// TIA Portal V20 export
FUNCTION "CallEnergyMeter" : Void   // FC9, LAD
TITLE = CALL_AIEnergyMeter_FC
AUTHOR : SICAR
FAMILY : Energy
VERSION : 1.0
// This block calls the blocks for the AI-Energy-management.
// For more informations see SICAR userdefined documentation / SICAR online-help.
// stored: IsIECCheckEnabled true, SetENOAutomatically true
   VAR_TEMP
      tempCommResourceCounter : Int;   // für FB-Aufruf: E2M_1500_AIEnergyMeter_DRV
      tempBitsHmi : "typeEnMeterBits";   // für FB-Aufruf: E2M_1500_AIEnergyMeter_DRV
   END_VAR
   // Ret_Val : Ret_Val
BEGIN

REGION Network 1: ChangeLog
   // SIEMENS AG / (c)Copyright 2023
   // ------------------------------------------------------------------------------
   // Title:            CallEnergyMeter (FC9)
   // Comment/Function: This block calls the blocks for the AI-Energy-management.
   // Library/Family:   Automation Framework
   // Author:           Siemens Digital Industry
   // Tested with:      ---
   // Engineering:      TIA Portal V19
   // Restrictions:     -
   // Requirements:     ---
   // ------------------------------------------------------------------------------
   // Change log table:
   // Version  | Date       | Expert in charge       | Changes applied
   // ---------|------------|------------------------|------------------------------
   // 05.00.00 | 01.09.2023 | SICAR
   //                         First released version
END_REGION

REGION Network 2: AI_EnergyMeter 1
   // Call of E2MenergyMeterDrv FB
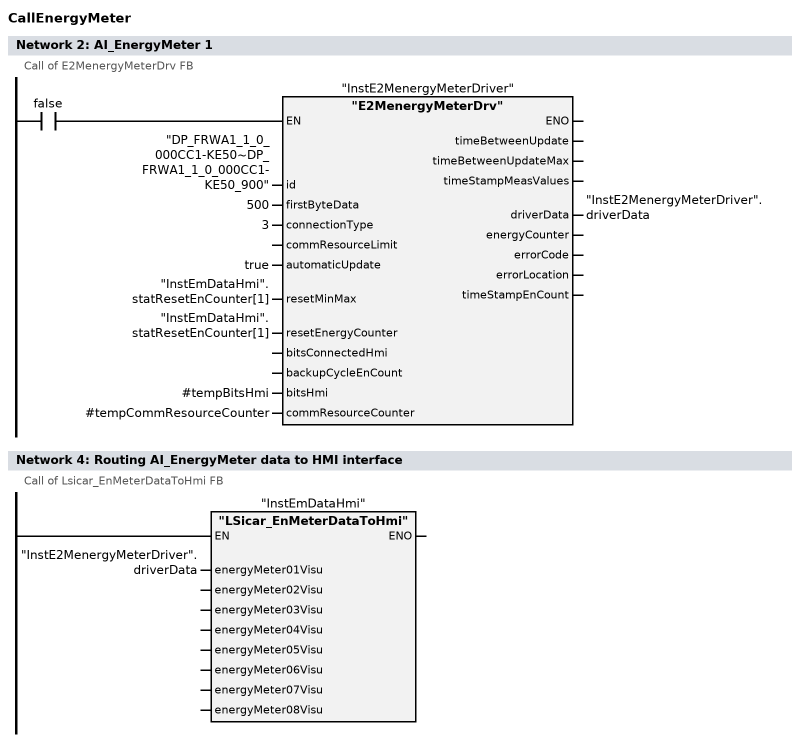
   RUNG wire#powerrail
      Contact( false )
      "InstE2MenergyMeterDriver"(id := "DP_FRWA1_1_0_000CC1-KE50~DP_FRWA1_1_0_000CC1-KE50_900", firstByteData := 500, connectionType := 3, commResourceLimit :=, automaticUpdate := true, resetMinMax := "InstEmDataHmi".statResetEnCounter[1], resetEnergyCounter := "InstEmDataHmi".statResetEnCounter[1], bitsConnectedHmi :=, backupCycleEnCount :=, bitsHmi := #tempBitsHmi, commResourceCounter := #tempCommResourceCounter, timeBetweenUpdate =>, timeBetweenUpdateMax =>, timeStampMeasValues =>, driverData => "InstE2MenergyMeterDriver".driverData, energyCounter =>, errorCode =>, errorLocation =>, timeStampEnCount =>)
   END_RUNG
   // the same network as SCL:
   IF false THEN
       "InstE2MenergyMeterDriver"(id := "DP_FRWA1_1_0_000CC1-KE50~DP_FRWA1_1_0_000CC1-KE50_900",   // "E2MenergyMeterDrv"
                               firstByteData := 500,
                               connectionType := 3,
                               automaticUpdate := true,
                               resetMinMax := "InstEmDataHmi".statResetEnCounter[1],
                               resetEnergyCounter := "InstEmDataHmi".statResetEnCounter[1],
                               bitsHmi := #tempBitsHmi,
                               commResourceCounter := #tempCommResourceCounter,
                               driverData => "InstE2MenergyMeterDriver".driverData);
   END_IF;
END_REGION

REGION Network 3 (SCL): Power meter

   // Voltage L-N
   "InstE2MenergyMeterDriver".driverData.uL1 := "PAC3220InPut"."Voltage_L1-N";
   "InstE2MenergyMeterDriver".driverData.uL2 := "PAC3220InPut"."Voltage_L2-N";
   "InstE2MenergyMeterDriver".driverData.uL3 := "PAC3220InPut"."Voltage_L3-N";
   "InstE2MenergyMeterDriver".driverData.uPhNaverage :=
   ("InstE2MenergyMeterDriver".driverData.uL1 + "InstE2MenergyMeterDriver".driverData.uL2 + "InstE2MenergyMeterDriver".driverData.uL3) / 3.0;

   IF "InstE2MenergyMeterDriver".driverData.uL1 < "InstE2MenergyMeterDriver".driverData.uL1Min OR "InstE2MenergyMeterDriver".driverData.uL1Min = 0.0 THEN
       "InstE2MenergyMeterDriver".driverData.uL1Min := "InstE2MenergyMeterDriver".driverData.uL1;
   END_IF;
   IF "InstE2MenergyMeterDriver".driverData.uL1 > "InstE2MenergyMeterDriver".driverData.uL1Max OR "InstE2MenergyMeterDriver".driverData.uL1Max = 0.0 THEN
       "InstE2MenergyMeterDriver".driverData.uL1Max := "InstE2MenergyMeterDriver".driverData.uL1;
   END_IF;

   IF "InstE2MenergyMeterDriver".driverData.uL2 < "InstE2MenergyMeterDriver".driverData.uL2Min OR "InstE2MenergyMeterDriver".driverData.uL2Min = 0.0 THEN
       "InstE2MenergyMeterDriver".driverData.uL2Min := "InstE2MenergyMeterDriver".driverData.uL2;
   END_IF;
   IF "InstE2MenergyMeterDriver".driverData.uL2 > "InstE2MenergyMeterDriver".driverData.uL2Max OR "InstE2MenergyMeterDriver".driverData.uL2Max = 0.0 THEN
       "InstE2MenergyMeterDriver".driverData.uL2Max := "InstE2MenergyMeterDriver".driverData.uL2;
   END_IF;

   IF "InstE2MenergyMeterDriver".driverData.uL3 < "InstE2MenergyMeterDriver".driverData.uL3Min OR "InstE2MenergyMeterDriver".driverData.uL3Min = 0.0 THEN
       "InstE2MenergyMeterDriver".driverData.uL3Min := "InstE2MenergyMeterDriver".driverData.uL3;
   END_IF;
   IF "InstE2MenergyMeterDriver".driverData.uL3 > "InstE2MenergyMeterDriver".driverData.uL3Max OR "InstE2MenergyMeterDriver".driverData.uL3Max = 0.0 THEN
       "InstE2MenergyMeterDriver".driverData.uL3Max := "InstE2MenergyMeterDriver".driverData.uL3;
   END_IF;

   IF "InstE2MenergyMeterDriver".driverData.uPhNaverage < "InstE2MenergyMeterDriver".driverData.uPhNaverageMin OR "InstE2MenergyMeterDriver".driverData.uPhNaverageMin = 0.0 THEN
       "InstE2MenergyMeterDriver".driverData.uPhNaverageMin := "InstE2MenergyMeterDriver".driverData.uPhNaverage;
   END_IF;
   IF "InstE2MenergyMeterDriver".driverData.uPhNaverage > "InstE2MenergyMeterDriver".driverData.uPhNaverageMax OR "InstE2MenergyMeterDriver".driverData.uPhNaverageMax = 0.0 THEN
       "InstE2MenergyMeterDriver".driverData.uPhNaverageMax := "InstE2MenergyMeterDriver".driverData.uPhNaverage;
   END_IF;

   // Voltage L-L
   "InstE2MenergyMeterDriver".driverData.uL1L2 := "PAC3220InPut"."Voltage_L1-L2";
   "InstE2MenergyMeterDriver".driverData.uL2L3 := "PAC3220InPut"."Voltage_L2-L3";
   "InstE2MenergyMeterDriver".driverData.uL3L1 := "PAC3220InPut"."Voltage_L3-L1";
   "InstE2MenergyMeterDriver".driverData.uPhPhAverage :=
   ("InstE2MenergyMeterDriver".driverData.uL1L2 + "InstE2MenergyMeterDriver".driverData.uL2L3 + "InstE2MenergyMeterDriver".driverData.uL3L1) / 3.0;

   IF "InstE2MenergyMeterDriver".driverData.uL1L2 < "InstE2MenergyMeterDriver".driverData.uL1L2Min OR "InstE2MenergyMeterDriver".driverData.uL1L2Min = 0.0 THEN
       "InstE2MenergyMeterDriver".driverData.uL1L2Min := "InstE2MenergyMeterDriver".driverData.uL1L2;
   END_IF;
   IF "InstE2MenergyMeterDriver".driverData.uL1L2 > "InstE2MenergyMeterDriver".driverData.uL1L2Max OR "InstE2MenergyMeterDriver".driverData.uL1L2Max = 0.0 THEN
       "InstE2MenergyMeterDriver".driverData.uL1L2Max := "InstE2MenergyMeterDriver".driverData.uL1L2;
   END_IF;

   IF "InstE2MenergyMeterDriver".driverData.uL2L3 < "InstE2MenergyMeterDriver".driverData.uL2L3Min OR "InstE2MenergyMeterDriver".driverData.uL2L3Min = 0.0 THEN
       "InstE2MenergyMeterDriver".driverData.uL2L3Min := "InstE2MenergyMeterDriver".driverData.uL2L3;
   END_IF;
   IF "InstE2MenergyMeterDriver".driverData.uL2L3 > "InstE2MenergyMeterDriver".driverData.uL2L3Max OR "InstE2MenergyMeterDriver".driverData.uL2L3Max = 0.0 THEN
       "InstE2MenergyMeterDriver".driverData.uL2L3Max := "InstE2MenergyMeterDriver".driverData.uL2L3;
   END_IF;

   IF "InstE2MenergyMeterDriver".driverData.uL3L1 < "InstE2MenergyMeterDriver".driverData.uL3L1Min OR "InstE2MenergyMeterDriver".driverData.uL3L1Min = 0.0 THEN
       "InstE2MenergyMeterDriver".driverData.uL3L1Min := "InstE2MenergyMeterDriver".driverData.uL3L1;
   END_IF;
   IF "InstE2MenergyMeterDriver".driverData.uL3L1 > "InstE2MenergyMeterDriver".driverData.uL3L1Max OR "InstE2MenergyMeterDriver".driverData.uL3L1Max = 0.0 THEN
       "InstE2MenergyMeterDriver".driverData.uL3L1Max := "InstE2MenergyMeterDriver".driverData.uL3L1;
   END_IF;

   IF "InstE2MenergyMeterDriver".driverData.uPhPhAverage < "InstE2MenergyMeterDriver".driverData.uPhPhAverageMin OR "InstE2MenergyMeterDriver".driverData.uPhPhAverageMin = 0.0 THEN
       "InstE2MenergyMeterDriver".driverData.uPhPhAverageMin := "InstE2MenergyMeterDriver".driverData.uPhPhAverage;
   END_IF;
   IF "InstE2MenergyMeterDriver".driverData.uPhPhAverage > "InstE2MenergyMeterDriver".driverData.uPhPhAverageMax OR "InstE2MenergyMeterDriver".driverData.uPhPhAverageMax = 0.0THEN
       "InstE2MenergyMeterDriver".driverData.uPhPhAverageMax := "InstE2MenergyMeterDriver".driverData.uPhPhAverage;
   END_IF;

   // Current
   "InstE2MenergyMeterDriver".driverData.iL1 := "PAC3220InPut".Current_L1;
   "InstE2MenergyMeterDriver".driverData.iL2 := "PAC3220InPut".Current_L2;
   "InstE2MenergyMeterDriver".driverData.iL3 := "PAC3220InPut".Current_L3;
   "InstE2MenergyMeterDriver".driverData.iAverage := "PAC3220InPut"."3-phase_average_current";

   IF "InstE2MenergyMeterDriver".driverData.iL1 < "InstE2MenergyMeterDriver".driverData.iL1Min OR "InstE2MenergyMeterDriver".driverData.iL1Min = 0.0 THEN
       "InstE2MenergyMeterDriver".driverData.iL1Min := "InstE2MenergyMeterDriver".driverData.iL1;
   END_IF;
   IF "InstE2MenergyMeterDriver".driverData.iL1 > "InstE2MenergyMeterDriver".driverData.iL1Max OR "InstE2MenergyMeterDriver".driverData.iL1Max = 0.0 THEN
       "InstE2MenergyMeterDriver".driverData.iL1Max := "InstE2MenergyMeterDriver".driverData.iL1;
   END_IF;

   IF "InstE2MenergyMeterDriver".driverData.iL2 < "InstE2MenergyMeterDriver".driverData.iL2Min OR "InstE2MenergyMeterDriver".driverData.iL2Min = 0.0 THEN
       "InstE2MenergyMeterDriver".driverData.iL2Min := "InstE2MenergyMeterDriver".driverData.iL2;
   END_IF;
   IF "InstE2MenergyMeterDriver".driverData.iL2 > "InstE2MenergyMeterDriver".driverData.iL2Max OR "InstE2MenergyMeterDriver".driverData.iL2Max = 0.0 THEN
       "InstE2MenergyMeterDriver".driverData.iL2Max := "InstE2MenergyMeterDriver".driverData.iL2;
   END_IF;

   IF "InstE2MenergyMeterDriver".driverData.iL3 < "InstE2MenergyMeterDriver".driverData.iL3Min OR "InstE2MenergyMeterDriver".driverData.iL3Min = 0.0 THEN
       "InstE2MenergyMeterDriver".driverData.iL3Min := "InstE2MenergyMeterDriver".driverData.iL3;
   END_IF;
   IF "InstE2MenergyMeterDriver".driverData.iL3 > "InstE2MenergyMeterDriver".driverData.iL3Max OR "InstE2MenergyMeterDriver".driverData.iL3Max = 0.0 THEN
       "InstE2MenergyMeterDriver".driverData.iL3Max := "InstE2MenergyMeterDriver".driverData.iL3;
   END_IF;

   IF "InstE2MenergyMeterDriver".driverData.iAverage < "InstE2MenergyMeterDriver".driverData.iAverageMin OR "InstE2MenergyMeterDriver".driverData.iAverageMin = 0.0 THEN
       "InstE2MenergyMeterDriver".driverData.iAverageMin := "InstE2MenergyMeterDriver".driverData.iAverage;
   END_IF;
   IF "InstE2MenergyMeterDriver".driverData.iAverage > "InstE2MenergyMeterDriver".driverData.iAverageMax OR "InstE2MenergyMeterDriver".driverData.iAverageMax = 0.0THEN
       "InstE2MenergyMeterDriver".driverData.iAverageMax := "InstE2MenergyMeterDriver".driverData.iAverage;
   END_IF;

   // Power factor
   "InstE2MenergyMeterDriver".driverData.cosL1 := "PAC3220InPut".Power_factor_L1;
   "InstE2MenergyMeterDriver".driverData.cosL2 := "PAC3220InPut".Power_factor_L2;
   "InstE2MenergyMeterDriver".driverData.cosL3 := "PAC3220InPut".Power_factor_L3;
   "InstE2MenergyMeterDriver".driverData.cosAverage := "PAC3220InPut".Total_power_factor;

   IF "InstE2MenergyMeterDriver".driverData.cosL1 < "InstE2MenergyMeterDriver".driverData.cosL1Min OR "InstE2MenergyMeterDriver".driverData.cosL1Min = 0.0 THEN
       "InstE2MenergyMeterDriver".driverData.cosL1Min := "InstE2MenergyMeterDriver".driverData.cosL1;
   END_IF;
   IF "InstE2MenergyMeterDriver".driverData.cosL1 > "InstE2MenergyMeterDriver".driverData.cosL1Max THEN
       "InstE2MenergyMeterDriver".driverData.cosL1Max := "InstE2MenergyMeterDriver".driverData.cosL1;
   END_IF;

   IF "InstE2MenergyMeterDriver".driverData.cosL2 < "InstE2MenergyMeterDriver".driverData.cosL2Min OR "InstE2MenergyMeterDriver".driverData.cosL2Min = 0.0 THEN
       "InstE2MenergyMeterDriver".driverData.cosL2Min := "InstE2MenergyMeterDriver".driverData.cosL2;
   END_IF;
   IF "InstE2MenergyMeterDriver".driverData.cosL2 > "InstE2MenergyMeterDriver".driverData.cosL2Max OR "InstE2MenergyMeterDriver".driverData.cosL2Max = 0.0 THEN
       "InstE2MenergyMeterDriver".driverData.cosL2Max := "InstE2MenergyMeterDriver".driverData.cosL2;
   END_IF;

   IF "InstE2MenergyMeterDriver".driverData.cosL3 < "InstE2MenergyMeterDriver".driverData.cosL3Min OR "InstE2MenergyMeterDriver".driverData.cosL3Min = 0.0 THEN
       "InstE2MenergyMeterDriver".driverData.cosL3Min := "InstE2MenergyMeterDriver".driverData.cosL3;
   END_IF;
   IF "InstE2MenergyMeterDriver".driverData.cosL3 > "InstE2MenergyMeterDriver".driverData.cosL3Max OR "InstE2MenergyMeterDriver".driverData.cosL3Max = 0.0THEN
       "InstE2MenergyMeterDriver".driverData.cosL3Max := "InstE2MenergyMeterDriver".driverData.cosL3;
   END_IF;

   IF "InstE2MenergyMeterDriver".driverData.cosAverage < "InstE2MenergyMeterDriver".driverData.cosAverageMin OR "InstE2MenergyMeterDriver".driverData.cosAverageMin = 0.0 THEN
       "InstE2MenergyMeterDriver".driverData.cosAverageMin := "InstE2MenergyMeterDriver".driverData.cosAverage;
   END_IF;
   IF "InstE2MenergyMeterDriver".driverData.cosAverage > "InstE2MenergyMeterDriver".driverData.cosAverageMax OR "InstE2MenergyMeterDriver".driverData.cosAverageMax = 0.0 THEN
       "InstE2MenergyMeterDriver".driverData.cosAverageMax := "InstE2MenergyMeterDriver".driverData.cosAverage;
   END_IF;

   // Frequency
   "InstE2MenergyMeterDriver".driverData.f := "PAC3220InPut".Line_frequency;

   IF "InstE2MenergyMeterDriver".driverData.f < "InstE2MenergyMeterDriver".driverData.fMin OR "InstE2MenergyMeterDriver".driverData.fMin = 0.0 THEN
       "InstE2MenergyMeterDriver".driverData.fMin := "InstE2MenergyMeterDriver".driverData.f;
   END_IF;
   IF "InstE2MenergyMeterDriver".driverData.f > "InstE2MenergyMeterDriver".driverData.fMax OR "InstE2MenergyMeterDriver".driverData.fMax = 0.0 THEN
       "InstE2MenergyMeterDriver".driverData.fMax := "InstE2MenergyMeterDriver".driverData.f;
   END_IF;


   // Apparent power
   "InstE2MenergyMeterDriver".driverData.sL1 := "Apparent power L1";
   "InstE2MenergyMeterDriver".driverData.sL2 := "Apparent power L2";
   "InstE2MenergyMeterDriver".driverData.sL3 := "Apparent power L3";
   "InstE2MenergyMeterDriver".driverData.sTotal := "PAC3220InPut".Total_apparent_power;

   IF "InstE2MenergyMeterDriver".driverData.sL1 < "InstE2MenergyMeterDriver".driverData.sL1Min OR "InstE2MenergyMeterDriver".driverData.sL1Min = 0.0 THEN
       "InstE2MenergyMeterDriver".driverData.sL1Min := "InstE2MenergyMeterDriver".driverData.sL1;
   END_IF;
   IF "InstE2MenergyMeterDriver".driverData.sL1 > "InstE2MenergyMeterDriver".driverData.sL1Max OR "InstE2MenergyMeterDriver".driverData.sL1Max = 0.0 THEN
       "InstE2MenergyMeterDriver".driverData.sL1Max := "InstE2MenergyMeterDriver".driverData.sL1;
   END_IF;

   IF "InstE2MenergyMeterDriver".driverData.sL2 < "InstE2MenergyMeterDriver".driverData.sL2Min OR "InstE2MenergyMeterDriver".driverData.sL2Min = 0.0 THEN
       "InstE2MenergyMeterDriver".driverData.sL2Min := "InstE2MenergyMeterDriver".driverData.sL2;
   END_IF;
   IF "InstE2MenergyMeterDriver".driverData.sL2 > "InstE2MenergyMeterDriver".driverData.sL2Max OR "InstE2MenergyMeterDriver".driverData.sL2Max = 0.0 THEN
       "InstE2MenergyMeterDriver".driverData.sL2Max := "InstE2MenergyMeterDriver".driverData.sL2;
   END_IF;

   IF "InstE2MenergyMeterDriver".driverData.sL3 < "InstE2MenergyMeterDriver".driverData.sL3Min OR "InstE2MenergyMeterDriver".driverData.sL3Min = 0.0 THEN
       "InstE2MenergyMeterDriver".driverData.sL3Min := "InstE2MenergyMeterDriver".driverData.sL3;
   END_IF;
   IF "InstE2MenergyMeterDriver".driverData.sL3 > "InstE2MenergyMeterDriver".driverData.sL3Max OR "InstE2MenergyMeterDriver".driverData.sL3Max = 0.0 THEN
       "InstE2MenergyMeterDriver".driverData.sL3Max := "InstE2MenergyMeterDriver".driverData.sL3;
   END_IF;

   IF "InstE2MenergyMeterDriver".driverData.sTotal < "InstE2MenergyMeterDriver".driverData.sTotalMin OR "InstE2MenergyMeterDriver".driverData.sTotalMin = 0.0 THEN
       "InstE2MenergyMeterDriver".driverData.sTotalMin := "InstE2MenergyMeterDriver".driverData.sTotal;
   END_IF;
   IF "InstE2MenergyMeterDriver".driverData.sTotal > "InstE2MenergyMeterDriver".driverData.sTotalMax OR "InstE2MenergyMeterDriver".driverData.sTotalMax = 0.0 THEN
       "InstE2MenergyMeterDriver".driverData.sTotalMax := "InstE2MenergyMeterDriver".driverData.sTotal;
   END_IF;

   // Active power
   "InstE2MenergyMeterDriver".driverData.pL1 := "Active power L1";
   "InstE2MenergyMeterDriver".driverData.pL2 := "Active power L2";
   "InstE2MenergyMeterDriver".driverData.pL3 := "Active power L3";
   "InstE2MenergyMeterDriver".driverData.pTotal := "PAC3220InPut".Total_active_power;

   IF "InstE2MenergyMeterDriver".driverData.pL1 < "InstE2MenergyMeterDriver".driverData.pL1Min OR "InstE2MenergyMeterDriver".driverData.pL1Min = 0.0 THEN
       "InstE2MenergyMeterDriver".driverData.pL1Min := "InstE2MenergyMeterDriver".driverData.pL1;
   END_IF;
   IF "InstE2MenergyMeterDriver".driverData.pL1 > "InstE2MenergyMeterDriver".driverData.pL1Max OR "InstE2MenergyMeterDriver".driverData.pL1Max = 0.0 THEN
       "InstE2MenergyMeterDriver".driverData.pL1Max := "InstE2MenergyMeterDriver".driverData.pL1;
   END_IF;

   IF "InstE2MenergyMeterDriver".driverData.pL2 < "InstE2MenergyMeterDriver".driverData.pL2Min OR "InstE2MenergyMeterDriver".driverData.pL2Min = 0.0 THEN
       "InstE2MenergyMeterDriver".driverData.pL2Min := "InstE2MenergyMeterDriver".driverData.pL2;
   END_IF;
   IF "InstE2MenergyMeterDriver".driverData.pL2 > "InstE2MenergyMeterDriver".driverData.pL2Max OR "InstE2MenergyMeterDriver".driverData.pL2Max = 0.0 THEN
       "InstE2MenergyMeterDriver".driverData.pL2Max := "InstE2MenergyMeterDriver".driverData.pL2;
   END_IF;

   IF "InstE2MenergyMeterDriver".driverData.pL3 < "InstE2MenergyMeterDriver".driverData.pL3Min OR "InstE2MenergyMeterDriver".driverData.pL3Min = 0.0 THEN
       "InstE2MenergyMeterDriver".driverData.pL3Min := "InstE2MenergyMeterDriver".driverData.pL3;
   END_IF;
   IF "InstE2MenergyMeterDriver".driverData.pL3 > "InstE2MenergyMeterDriver".driverData.pL3Max OR "InstE2MenergyMeterDriver".driverData.pL3Max = 0.0 THEN
       "InstE2MenergyMeterDriver".driverData.pL3Max := "InstE2MenergyMeterDriver".driverData.pL3;
   END_IF;

   IF "InstE2MenergyMeterDriver".driverData.pTotal < "InstE2MenergyMeterDriver".driverData.pTotalMin OR "InstE2MenergyMeterDriver".driverData.pTotalMin = 0.0 THEN
       "InstE2MenergyMeterDriver".driverData.pTotalMin := "InstE2MenergyMeterDriver".driverData.pTotal;
   END_IF;
   IF "InstE2MenergyMeterDriver".driverData.pTotal > "InstE2MenergyMeterDriver".driverData.pTotalMax OR "InstE2MenergyMeterDriver".driverData.pTotalMax = 0.0 THEN
       "InstE2MenergyMeterDriver".driverData.pTotalMax := "InstE2MenergyMeterDriver".driverData.pTotal;
   END_IF;

   // Reactive power
   "InstE2MenergyMeterDriver".driverData.qL1 := "Reactive power L1";
   "InstE2MenergyMeterDriver".driverData.qL2 := "Reactive power L2";
   "InstE2MenergyMeterDriver".driverData.qL3 := "Reactive power L3";
   "InstE2MenergyMeterDriver".driverData.qTotal := "PAC3220InPut"."Total_reactive_power_(VARn)";

   IF "InstE2MenergyMeterDriver".driverData.qL1 < "InstE2MenergyMeterDriver".driverData.qL1Min OR "InstE2MenergyMeterDriver".driverData.qL1Min = 0.0 THEN
       "InstE2MenergyMeterDriver".driverData.qL1Min := "InstE2MenergyMeterDriver".driverData.qL1;
   END_IF;
   IF "InstE2MenergyMeterDriver".driverData.qL1 > "InstE2MenergyMeterDriver".driverData.qL1Max OR "InstE2MenergyMeterDriver".driverData.qL1Max = 0.0 THEN
       "InstE2MenergyMeterDriver".driverData.qL1Max := "InstE2MenergyMeterDriver".driverData.qL1;
   END_IF;

   IF "InstE2MenergyMeterDriver".driverData.qL2 < "InstE2MenergyMeterDriver".driverData.qL2Min OR "InstE2MenergyMeterDriver".driverData.qL2Min = 0.0 THEN
       "InstE2MenergyMeterDriver".driverData.qL2Min := "InstE2MenergyMeterDriver".driverData.qL2;
   END_IF;
   IF "InstE2MenergyMeterDriver".driverData.qL2 > "InstE2MenergyMeterDriver".driverData.qL2Max OR "InstE2MenergyMeterDriver".driverData.qL2Max = 0.0 THEN
       "InstE2MenergyMeterDriver".driverData.qL2Max := "InstE2MenergyMeterDriver".driverData.qL2;
   END_IF;

   IF "InstE2MenergyMeterDriver".driverData.qL3 < "InstE2MenergyMeterDriver".driverData.qL3Min OR "InstE2MenergyMeterDriver".driverData.qL3Min = 0.0 THEN
       "InstE2MenergyMeterDriver".driverData.qL3Min := "InstE2MenergyMeterDriver".driverData.qL3;
   END_IF;
   IF "InstE2MenergyMeterDriver".driverData.qL3 > "InstE2MenergyMeterDriver".driverData.qL3Max OR "InstE2MenergyMeterDriver".driverData.qL3Max = 0.0 THEN
       "InstE2MenergyMeterDriver".driverData.qL3Max := "InstE2MenergyMeterDriver".driverData.qL3;
   END_IF;

   IF "InstE2MenergyMeterDriver".driverData.qTotal < "InstE2MenergyMeterDriver".driverData.qTotalMin OR "InstE2MenergyMeterDriver".driverData.qTotalMin = 0.0 THEN
       "InstE2MenergyMeterDriver".driverData.qTotalMin := "InstE2MenergyMeterDriver".driverData.qTotal;
   END_IF;
   IF "InstE2MenergyMeterDriver".driverData.qTotal > "InstE2MenergyMeterDriver".driverData.qTotalMax OR "InstE2MenergyMeterDriver".driverData.qTotalMax = 0.0 THEN
       "InstE2MenergyMeterDriver".driverData.qTotalMax := "InstE2MenergyMeterDriver".driverData.qTotal;
   END_IF;

   // Energy Tarif
   "InstE2MenergyMeterDriver".driverData.eActiveRate1Import := "Active energy import tariff 1(F)";
   "InstE2MenergyMeterDriver".driverData.eReactiveRate1Import := "Reactive energy import tariff 1 (F)";
   "InstE2MenergyMeterDriver".driverData.eApparentRate1Import := "Apparent energy tariff 1 (F)";
   "InstE2MenergyMeterDriver".driverData.eActiveRate1Export := "Active energy export tariff 1(F)";
   "InstE2MenergyMeterDriver".driverData.eReactiveRate1Export := "Reactive energy export tariff 1 (F)";






   // Reset 
   IF "InstEmDataHmi".statResetMinMaxAll  THEN

       // 모든 Min/Max 초기화 (Actual 값으로)
       "InstE2MenergyMeterDriver".driverData.uL1Min := 0.0;
       "InstE2MenergyMeterDriver".driverData.uL1Max := 0.0;
       "InstE2MenergyMeterDriver".driverData.uL2Min := 0.0;
       "InstE2MenergyMeterDriver".driverData.uL2Max := 0.0;
       "InstE2MenergyMeterDriver".driverData.uL3Min := 0.0;
       "InstE2MenergyMeterDriver".driverData.uL3Max := 0.0;

       "InstE2MenergyMeterDriver".driverData.uL1L2Min := 0.0;
       "InstE2MenergyMeterDriver".driverData.uL1L2Max := 0.0;
       "InstE2MenergyMeterDriver".driverData.uL2L3Min := 0.0;
       "InstE2MenergyMeterDriver".driverData.uL2L3Max := 0.0;
       "InstE2MenergyMeterDriver".driverData.uL3L1Min := 0.0;
       "InstE2MenergyMeterDriver".driverData.uL3L1Max := 0.0;

       "InstE2MenergyMeterDriver".driverData.uPhNaverageMin := 0.0;
       "InstE2MenergyMeterDriver".driverData.uPhNaverageMax := 0.0;

       "InstE2MenergyMeterDriver".driverData.uPhPhAverageMin := 0.0;
       "InstE2MenergyMeterDriver".driverData.uPhPhAverageMax := 0.0;

       "InstE2MenergyMeterDriver".driverData.iL1Min := 0.0;
       "InstE2MenergyMeterDriver".driverData.iL1Max := 0.0;
       "InstE2MenergyMeterDriver".driverData.iL2Min := 0.0;
       "InstE2MenergyMeterDriver".driverData.iL2Max := 0.0;
       "InstE2MenergyMeterDriver".driverData.iL3Min := 0.0;
       "InstE2MenergyMeterDriver".driverData.iL3Max := 0.0;

       "InstE2MenergyMeterDriver".driverData.iAverageMin := 0.0;
       "InstE2MenergyMeterDriver".driverData.iAverageMax := 0.0;

       "InstE2MenergyMeterDriver".driverData.cosL1Min := 0.0;
       "InstE2MenergyMeterDriver".driverData.cosL1Max := 0.0;
       "InstE2MenergyMeterDriver".driverData.cosL2Min := 0.0;
       "InstE2MenergyMeterDriver".driverData.cosL2Max := 0.0;
       "InstE2MenergyMeterDriver".driverData.cosL3Min := 0.0;
       "InstE2MenergyMeterDriver".driverData.cosL3Max := 0.0;

       "InstE2MenergyMeterDriver".driverData.cosAverageMin := 0.0;
       "InstE2MenergyMeterDriver".driverData.cosAverageMax := 0.0;

       "InstE2MenergyMeterDriver".driverData.fMin := 0.0;
       "InstE2MenergyMeterDriver".driverData.fMax := 0.0;

       "InstE2MenergyMeterDriver".driverData.pTotalMin := 0.0;
       "InstE2MenergyMeterDriver".driverData.pTotalMax := 0.0;
       "InstE2MenergyMeterDriver".driverData.qTotalMin := 0.0;
       "InstE2MenergyMeterDriver".driverData.qTotalMax := 0.0;
       "InstE2MenergyMeterDriver".driverData.sTotalMin := 0.0;
       "InstE2MenergyMeterDriver".driverData.sTotalMax := 0.0;

       "InstE2MenergyMeterDriver".driverData.sL1Min := 0.0;
       "InstE2MenergyMeterDriver".driverData.sL1Max := 0.0;
       "InstE2MenergyMeterDriver".driverData.sL2Min := 0.0;
       "InstE2MenergyMeterDriver".driverData.sL2Max := 0.0;
       "InstE2MenergyMeterDriver".driverData.sL3Min := 0.0;
       "InstE2MenergyMeterDriver".driverData.sL3Max := 0.0;

       "InstE2MenergyMeterDriver".driverData.pL1Min := 0.0;
       "InstE2MenergyMeterDriver".driverData.pL1Max := 0.0;
       "InstE2MenergyMeterDriver".driverData.pL2Min := 0.0;
       "InstE2MenergyMeterDriver".driverData.pL2Max := 0.0;
       "InstE2MenergyMeterDriver".driverData.pL3Min := 0.0;
       "InstE2MenergyMeterDriver".driverData.pL3Max := 0.0;

       "InstE2MenergyMeterDriver".driverData.qL1Min := 0.0;
       "InstE2MenergyMeterDriver".driverData.qL1Max := 0.0;
       "InstE2MenergyMeterDriver".driverData.qL2Min := 0.0;
       "InstE2MenergyMeterDriver".driverData.qL2Max := 0.0;
       "InstE2MenergyMeterDriver".driverData.qL3Min := 0.0;
       "InstE2MenergyMeterDriver".driverData.qL3Max := 0.0;

   END_IF;
END_REGION

REGION Network 4: Routing AI_EnergyMeter data to HMI interface
   // Call of Lsicar_EnMeterDataToHmi FB
   RUNG wire#powerrail
      "InstEmDataHmi"(energyMeter01Visu := "InstE2MenergyMeterDriver".driverData, energyMeter02Visu :=, energyMeter03Visu :=, energyMeter04Visu :=, energyMeter05Visu :=, energyMeter06Visu :=, energyMeter07Visu :=, energyMeter08Visu :=)
   END_RUNG
   // the same network as SCL:
   "InstEmDataHmi"(energyMeter01Visu := "InstE2MenergyMeterDriver".driverData);   // "LSicar_EnMeterDataToHmi"
END_REGION
END_FUNCTION
